// TIA Portal project "Biegewerkzeug_0" (V20)

(* hardware
DEVICE "S7-300/ET200M-Station_1"  S7-300 station
   slot 0: "Profilschiene_0"  Rail  6ES7 390-1***0-0AA0
   slot 2: "PLC_1"  CPU 315-2 PN/DP  6ES7 315-2EH14-0AB0  V3.2.18
      slot 2: "PROFINET-Schnittstelle_1"  PN-IO
         slot 1: "Port_1"  Port
         slot 2: "Port_2"  Port
   slot 4: "DI 16x24VDC_1"  DI16 x 24VDC, interrupt  6ES7 321-7BH01-0AB0
   slot 5: "DO 8x24VDC/0.5A_1"  DO8 x 24VDC / 0.5A  6ES7 322-8BF00-0AB0
*)

// ===== PLC "PLC_1"  CPU 315-2 PN/DP =====

VAR_GLOBAL   // PLC tag table "Standard-Variablentabelle"
   "S1" AT %E0.7 : Bool;
   "1B1" AT %E0.0 : Bool;
   "1B2" AT %E0.1 : Bool;
   "2B1" AT %E1.0 : Bool;
   "2B2" AT %E1.1 : Bool;
   "1M1" AT %A0.0 : Bool;
   "2M1" AT %A1.0 : Bool;
   "Prozessstart" AT %M0.0 : Bool;
   "Spule 1 aktiv" AT %M0.1 : Bool;
   "Spule 2 aktiv" AT %M0.2 : Bool;
   "Prozessende" AT %M0.3 : Bool;
END_VAR

DATA_BLOCK "Biegewerkzeug_0_DB"   // DB1
{ S7_Optimized_Access := 'FALSE' }
VERSION : 0.1
// stored: InstanceOfName Biegewerkzeug_0
"Biegewerkzeug_0"
BEGIN
END_DATA_BLOCK

FUNCTION_BLOCK "Biegewerkzeug_0"   // FB1, FBD
{ S7_Optimized_Access := 'FALSE' }
VERSION : 0.1
BEGIN

REGION Network 1: Prozesstart
   // Nach Betätigung des Tasters-S1 wird hier der Prozess gestartet. Ein erneuter Start ist erst nach Rücksetzen durch "Prozessende" möglich.
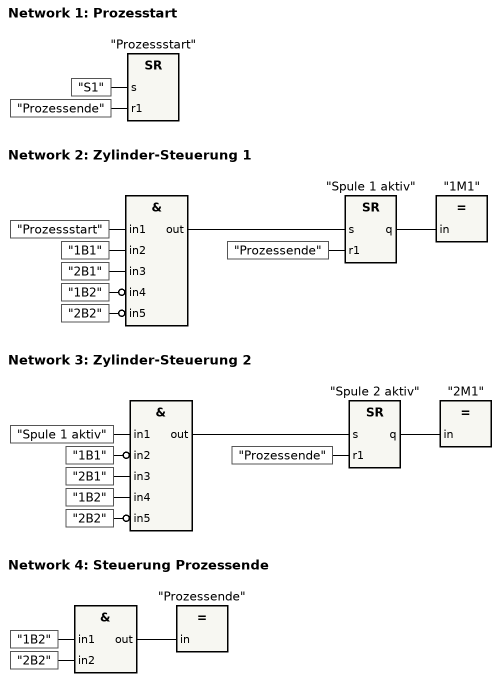
   IF "S1" THEN
       "Prozessstart" := TRUE;   // SR flip-flop
   END_IF;
   IF "Prozessende" THEN "Prozessstart" := FALSE; END_IF;
END_REGION

REGION Network 2: Zylinder-Steuerung 1
   // Wenn der Prozess gestartet werden soll und beide Kolben eingefahren sind, dann schalte die 1. Spule ein, wodurch Kolben 1 ausgefahren wird.
   IF "Prozessstart" AND "1B1" AND "2B1" AND NOT "1B2" AND NOT "2B2" THEN
       "Spule 1 aktiv" := TRUE;   // SR flip-flop
   END_IF;
   IF "Prozessende" THEN "Spule 1 aktiv" := FALSE; END_IF;
   "1M1" := "Spule 1 aktiv";
END_REGION

REGION Network 3: Zylinder-Steuerung 2
   // Wenn Spannung auf Spule 1 ist und dadurch der 1. Kolben komplett ausgefahren wurde und Kolben 2 unverändert ist, dann schalte die 2. Spule ein, wodurch Kolben 2 ausgefahren wird.
   IF "Spule 1 aktiv" AND NOT "1B1" AND "2B1" AND "1B2" AND NOT "2B2" THEN
       "Spule 2 aktiv" := TRUE;   // SR flip-flop
   END_IF;
   IF "Prozessende" THEN "Spule 2 aktiv" := FALSE; END_IF;
   "2M1" := "Spule 2 aktiv";
END_REGION

REGION Network 4: Steuerung Prozessende
   // Wenn beide Spulen aktiv sind und dadurch beide Kolben die Endstellung erreicht haben setze Merker "Prozessende". Dieser setzt die beide Spulen und den Taster-S1 für einen erneuten Start des Prozesses zurück.
   "Prozessende" := "1B2" AND "2B2";
END_REGION
END_FUNCTION_BLOCK

ORGANIZATION_BLOCK "Main"   // OB1, FBD
TITLE = "Main Program Sweep (Cycle)"
{ S7_Optimized_Access := 'FALSE' }
VERSION : 0.1
   VAR_TEMP
      OB1_EV_CLASS : Byte;   // Bits 0-3 = 1 (Coming event), Bits 4-7 = 1 (Event class 1)
      OB1_SCAN_1 : Byte;   // 1 (Cold restart scan 1 of OB 1), 3 (Scan 2-n of OB 1)
      OB1_PRIORITY : Byte;   // Priority of OB Execution
      OB1_OB_NUMBR : Byte;   // 1 (Organization block 1, OB1)
      OB1_RESERVED_1 : Byte;   // Reserved for system
      OB1_RESERVED_2 : Byte;   // Reserved for system
      OB1_PREV_CYCLE : Int;   // Cycle time of previous OB1 scan (milliseconds)
      OB1_MIN_CYCLE : Int;   // Minimum cycle time of OB1 (milliseconds)
      OB1_MAX_CYCLE : Int;   // Maximum cycle time of OB1 (milliseconds)
      OB1_DATE_TIME : Date_And_Time;   // Date and time OB1 started
   END_VAR
BEGIN

REGION Network 1
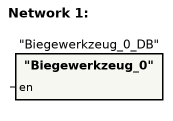
   "Biegewerkzeug_0_DB"();   // "Biegewerkzeug_0"
END_REGION
END_ORGANIZATION_BLOCK